# EPICS StreamDevice protocol: streamDevice/bennett.proto
# Bennett's Sidekick EPICS protocol file
# Built by examining examples at: https://paulscherrerinstitute.github.io/StreamDevice/protocol.html#gen

Terminator = CR LF;

info {
	ExtraInput = Ignore;
	out "*IDN?";
	in "%39c";
}

debug {
   ExtraInput = Ignore;
   out "%s";
   in "%39c";
}

# Queryable and settable
SpeakerShutdownQ {
    out "SPEAker:SHUTdown?";
    in "%i";
}

SpeakerShutdown {
    out "SPEAker:SHUTdown %i";
    @init { SpeakerShutdownQ; }
}

SpeakerMuteQ {
    out "SPEAker:MUTE?";
    in "%i";
}

SpeakerMute {
    out "SPEAker:MUTE %i";
    @init { SpeakerMuteQ; }
}

SpeakerVolumeQ {
    out "SPEAker:VOLume?";
    in "%u";
}

SpeakerVolume {
    out "SPEAker:VOLume %u";
    @init { SpeakerVolumeQ; }
}

# Settable only
SpeakerPlay {
    out "SPEAker:PLAY";
}
